(*			
	RAFALOS
	Rafał Osajda		23.09.2025		TC 4024.66
	Struktura pomocnicza potrzeba do wiazania zmiennych
*)
TYPE ST_BaseHMITopElement_View_Link :
STRUCT
	stLoggerElement				: ST_BaseHMILoggerElement_View;
	stComponent					: ST_BaseHMIComponent_View;
	stControlElement			: ST_BaseHMIControlElement_View;
	stGroupElement				: ST_BaseHMIGroupElement_View;
	stTopElement				: ST_BaseHMITopElement_View;
END_STRUCT
END_TYPE

(* stored: Version 1.1.0.1
   DUT ST_BaseHMITopElement_View_Link: Id {533e9167-bcb7-04ba-2414-b4dc5f61b55b} *)
